{attribute 'qualified_only'}
VAR_GLOBAL
TYPE
	CLAMP_STATE: (e_OPEN, e_CLOSED_FULL, e_CLOSED, e_ERROR);
END_TYPE		

END_VAR

(* stored: Version 1.1.0.1, ProductVersion 3.1.4024.0
   GVL CLAMP_STATE: Id {7b75da27-6950-4b61-8247-fae8d6f4ad07} *)
